# EPICS substitutions: db/Beckhoff_5XXX/ecmcEL5102.substitutions
file "ecmcEL51xx-32bit-chX.template"
{
    pattern {CH_ID}
            {01   }
            {02   }
}
